// TIA Portal V19 export
DATA_BLOCK "DB_RecipeEmpty"   // DB51
{ S7_Optimized_Access := 'TRUE' }
// stored: AutoNumber false, MemoryReserve 100
   VAR
      RecipeEmpty { ExternalAccessible := 'False'; ExternalVisible := 'False'; ExternalWritable := 'False'} : "stRecipe";
   END_VAR
BEGIN
   RecipeEmpty.RecipeLayerType[1].RecipeLayerTypeName := 'Putty';
   RecipeEmpty.RecipeLayerType[1].JobTableLeft[0].SetForceZero := 0;
   RecipeEmpty.RecipeLayerType[2].JobTableLeft[0].SetForceZero := 0;
   RecipeEmpty.RecipeLayerType[1].JobTableLeft[0].SetForceTarget := 0;
   RecipeEmpty.RecipeLayerType[2].JobTableLeft[0].SetForceTarget := 0;
   RecipeEmpty.RecipeLayerType[1].JobTableLeft[0].SetTimeRamp := 0;
   RecipeEmpty.RecipeLayerType[2].JobTableLeft[0].SetTimeRamp := 0;
   RecipeEmpty.RecipeLayerType[1].JobTableLeft[0].SetSpeed := 0;
   RecipeEmpty.RecipeLayerType[2].JobTableLeft[0].SetSpeed := 0;
   RecipeEmpty.RecipeLayerType[1].JobTableLeft[0].SetRobotSpeed := 0;
   RecipeEmpty.RecipeLayerType[2].JobTableLeft[0].SetRobotSpeed := 0;
   RecipeEmpty.RecipeLayerType[1].JobTableLeft[0].WornPaperDistance := 0;
   RecipeEmpty.RecipeLayerType[2].JobTableLeft[0].WornPaperDistance := 0;
   RecipeEmpty.RecipeLayerType[1].JobTableLeft[0].Gimball := 0;
   RecipeEmpty.RecipeLayerType[2].JobTableLeft[0].Gimball := 0;
   RecipeEmpty.RecipeLayerType[1].JobTableRight[0].SetForceZero := 0;
   RecipeEmpty.RecipeLayerType[2].JobTableRight[0].SetForceZero := 0;
   RecipeEmpty.RecipeLayerType[1].JobTableRight[0].SetForceTarget := 0;
   RecipeEmpty.RecipeLayerType[2].JobTableRight[0].SetForceTarget := 0;
   RecipeEmpty.RecipeLayerType[1].JobTableRight[0].SetTimeRamp := 0;
   RecipeEmpty.RecipeLayerType[2].JobTableRight[0].SetTimeRamp := 0;
   RecipeEmpty.RecipeLayerType[1].JobTableRight[0].SetSpeed := 0;
   RecipeEmpty.RecipeLayerType[2].JobTableRight[0].SetSpeed := 0;
   RecipeEmpty.RecipeLayerType[1].JobTableRight[0].SetRobotSpeed := 0;
   RecipeEmpty.RecipeLayerType[2].JobTableRight[0].SetRobotSpeed := 0;
   RecipeEmpty.RecipeLayerType[1].JobTableRight[0].WornPaperDistance := 0;
   RecipeEmpty.RecipeLayerType[2].JobTableRight[0].WornPaperDistance := 0;
   RecipeEmpty.RecipeLayerType[1].JobTableRight[0].Gimball := 0;
   RecipeEmpty.RecipeLayerType[2].JobTableRight[0].Gimball := 0;
END_DATA_BLOCK
